Staubli VAL3: MotionPage.pjx

--- MotionPage.pjx ---
Parameters version=s7.1.3 stackSize=5000 millimeterUnit=true
Program file=Align.pgx
Program file=AlignPage.pgx
Program file=BackHome.pgx
Program file=BackHomePage.pgx
Program file=CompareJoint.pgx
Program file=ComparePoint.pgx
Program file=setAxis.pgx
Program file=start.pgx
Program file=stop.pgx
Data file=MotionPage.dtx
Library alias=user path=Disk://userPage/userPage.pjx

--- AlignPage.pgx ---
public program AlignPage(tool x_tTool)
  local num l_nKey
  local string l_sButton[2]
  local num l_i
  local bool l_bAlignDone
  local bool l_bExit
  local string l_sYesNo
begin
  //-----------------------------------------------------------------------
  //Header begin
  //Description of program
  //  工具对齐界面
  //  F1:终止
  //Input parameters
  //  tool x_tTool:工具值
  //Output paramaters
  //Example
  //  call Align(tool)
  //History
  //  Creation : 2012-06-11 - PF.Zhong
  //Header end
  //-----------------------------------------------------------------------
  cls()
  bAlignDone=false
  l_bExit=false
  taskCreate "Align",30,Align(x_tTool,bAlignDone)
  delay(0.1)
  while !bAlignDone and !l_bExit
      call user:timerDialog("机器人工具头正在对齐，请按住Move/Hold键",0)
      call user:typeLen(1,13,"终止",4)
      l_nKey=getKey()
      switch l_nKey
        case 271
          //终止
          cls()
          l_sButton[0]="是"
          l_sButton[1]="否"
          call user:questionDialog("是否终止对齐?",l_sButton,l_i)
          if l_i==0 or l_i==1
            resetMotion()
            stopMove()
            taskKill("Align")
            l_bExit=true
          else
            cls()
          endIf
        break
      endSwitch
      delay(0)
  endWhile
  if bAlignDone
    l_sYesNo="确定"
    call user:yes("对齐完毕!",l_sYesNo)
  else
    l_sYesNo="确定"
    call user:yes("对齐未完成!",l_sYesNo)
  endIf
end

--- CompareJoint.pgx ---
public program CompareJoint(joint x_jJoint1, joint x_jJoint2, bool& x_bSame, num x_nAixNum)
begin
  //-----------------------------------------------------------------------
  //Header begin
  //Description of program
  //  判断手臂是否在指定关节位置
  //Input parameters
  //  joint x_jJoint:关节位置
  //Output paramaters
  //  bool x_bHome:是否在指定关节位置
  //Example
  //  call TestHome(bOK,joint)
  //History
  //  Creation : 2012-06-11 - PF.Zhong
  //Header end
  //-----------------------------------------------------------------------
  switch x_nAixNum
    //六轴
    case 6
      if abs(x_jJoint1.j1-x_jJoint2.j1)<0.02
        if abs(x_jJoint1.j2-x_jJoint2.j2)<0.02
          if abs(x_jJoint1.j3-x_jJoint2.j3)<0.02
            if abs(x_jJoint1.j4-x_jJoint2.j4)<0.02
              if abs(x_jJoint1.j5-x_jJoint2.j5)<0.02
                if abs(x_jJoint1.j6-x_jJoint2.j6)<0.02
                  x_bSame=true
                else
                  x_bSame=false
                endIf
              else
                x_bSame=false
              endIf
            else
              x_bSame=false
            endIf
          else
            x_bSame=false
          endIf
        else
          x_bSame=false
        endIf
      else
        x_bSame=false
      endIf
    break
    //四轴
    case 4
      if abs(x_jJoint1.j1-x_jJoint2.j1)<0.02
        if abs(x_jJoint1.j2-x_jJoint2.j2)<0.02
          if abs(x_jJoint1.j3-x_jJoint2.j3)<0.02
            if abs(x_jJoint1.j4-x_jJoint2.j4)<0.02
            else
              x_bSame=false
            endIf
          else
            x_bSame=false
          endIf
        else
          x_bSame=false
        endIf
      else
        x_bSame=false
      endIf
    break
  endSwitch
end

--- ComparePoint.pgx ---
public program ComparePoint(pointRx& x_pPoint1, point& x_pPoint2, bool& x_bSame)
  local trsf l_trTrsf1
  local trsf l_trTrsf2
begin
  //比较两个点
  l_trTrsf1=position(x_pPoint1,world)
  l_trTrsf2=position(x_pPoint2,world)
  if abs(l_trTrsf1.x-l_trTrsf2.x)<0.05
    if abs(l_trTrsf1.y-l_trTrsf2.y)<0.05
      if abs(l_trTrsf1.z-l_trTrsf2.z)<0.05
        if abs(l_trTrsf1.rx-l_trTrsf2.rx)<0.05
          if abs(l_trTrsf1.ry-l_trTrsf2.ry)<0.05
            if abs(l_trTrsf1.rz-l_trTrsf2.rz)<0.05
              x_bSame=true
              return
            else
              x_bSame=false
              return
            endIf
          else
            x_bSame=false
            return
          endIf
        else
          x_bSame=false
          return
        endIf
      else
        x_bSame=false
        return
      endIf
    else
      x_bSame=false
      return
    endIf
  else
    x_bSame=false
    return
  endIf
end
